Fanuc KAREL source: kt00753.KL

-- PROVISIONAL review KL for V770-1; original PC SHA256 f040237fa62705f4eac64bebdba3df519ead179c07ae2e84cc107083601a8596
-- Incomplete behavior may be omitted. Consult companion uncertainty JSON. Do not deploy.
PROGRAM KT00753
%NOLOCKGROUP
VAR
  OUT : REAL
-- UNRESOLVED_DECL Y1 type=002018
-- UNRESOLVED_DECL Y2 type=002018
BEGIN
  -- UNRESOLVED_PC offsets 5-19; opcodes 2E,22,9D,33,B2
  -- UNRESOLVED_PC offsets 24-38; opcodes 2E,22,9D,33,B2
  -- UNRESOLVED_PC offsets 43-57; opcodes 2E,22,9D,33,B2
  -- UNRESOLVED_PC offsets 62-76; opcodes 2E,22,9D,33,B2
  -- UNRESOLVED_PC offsets 81-98; opcodes 22,9D,33,B1,50,64,23
  -- UNRESOLVED_PC offsets 103-107; opcodes 7F
END KT00753
